Staubli VAL3: OMAC_Abort.pgx

program OMAC_Abort()
begin
  //OMAC进程:aborting
  _nOmacStat=10
  logMsg("上位机手动操作：急停")
  resetMotion()
  stopMove()

  call setAlarm(10)
  // Stop task

  taskKill("cellManager")
  taskKill("overflowPick")
  taskKill("productionCycle")
  taskKill("Reset")
  taskKill("Start")
  taskKill("Hold")
  taskKill("Unhold")
  taskKill("Stop")
  taskKill("TransferQueue1")
  taskKill("robot2PLC")
  taskKill("robot2PC")

  wait(isSettled())
  wait(taskStatus("Reset")==-1)
  wait(taskStatus("Start")==-1)
  wait(taskStatus("Hold")==-1)
  wait(taskStatus("Unhold")==-1)
  wait(taskStatus("Stop")==-1)
  wait(taskStatus("cellManager")==-1)
  wait(taskStatus("TransferQueue1")==-1)
  wait(taskStatus("overflowPick")==-1)
  wait(taskStatus("productionCycle")==-1)

  if _bConvExist
    call mot:kill()
    _bConvExist=false
  endIf
  disablePower()
  wait(isPowered()==false)
  //OMAC进程:Stopped
  _nOmacStat=9
  delay(0)
end
